(* Logix 5000 project; controller Heat_circuit_control Emulate 5570 rev 30.12; software revision 30.01 *)

TASK MainTask (continuous, watchdog 500 ms) : MainProgram

MODULES
   Local : Emulate 5570 (ICP 3, rev 30.12)
      HOA_Digital_module : 1756-IB16 (ICP 2, rev 3.1, Input RPI 20 ms)
      Alarm_digital_output : vendor 1 type 7 code 18 (ICP 4, rev 3.1, Output RPI 20 ms)
      Analog_Valve_control : vendor 1 type 10 code 114 (ICP 0, rev 2.1, Input RPI 100 ms)
      Analog_Temperature_Output : vendor 1 type 10 code 115 (ICP 1, rev 2.1, Output RPI 25 ms)
END_MODULES

VAR_GLOBAL   (* controller tags *)
   Auto_control : ALIAS FOR Local:2:I.Data.2;
   Hand_control : ALIAS FOR Local:2:I.Data.0;
   Off_control : ALIAS FOR Local:2:I.Data.1;
   Solenoid_Valve : ALIAS FOR Local:0:I.Ch1Data;
   Temperature_level : ALIAS FOR Local:1:O.Ch1Data;
END_VAR

PROGRAM MainProgram   (* main routine MainRoutine *)
VAR
   Alarm : ALIAS FOR Local:4:O.Data.1;
   alarm_on : BOOL;
   Alarm_reset : ALIAS FOR Local:4:O.Data.0;
   alarm_timer : TIMER := (PRE := 5000);
   auto : BOOL;
   auto_mode : BOOL;
   check_timer : TIMER := (PRE := 5000);
   checking_light : BOOL;
   close_bit : BOOL;
   count : COUNTER;
   danger_bit : BOOL;
   high_limit : REAL;
   HOA : DINT;
   low_point : REAL;
   Manual : BOOL;
   Notification : ALIAS FOR Local:4:O.Data.2;
   OFF : BOOL;
   ons : BOOL;
   ons_10 : BOOL;
   ons_2 : BOOL;
   ons_3 : BOOL;
   ons_9 : BOOL;
   open_bit : BOOL;
   Openning : REAL;
   Set_Point : REAL;
   Solenoid_Valve_1 : REAL;
   Sub_light : BOOL;
   Timer_wait : TIMER := (PRE := 5000);
   Timer_wait_2 : TIMER := (PRE := 5000);
   Total : REAL;
   transfer : REAL;
   TT : BOOL;
   TT_2 : BOOL;
   TT_3 : BOOL;
   TT_4 : BOOL;
   user_input : REAL;
   user_val : REAL;
   value : REAL;
   wait_timer : TIMER := (PRE := 5000);
   wait_timer_2 : TIMER := (PRE := 5000);
END_VAR

ROUTINE Alarm   (* ladder *)
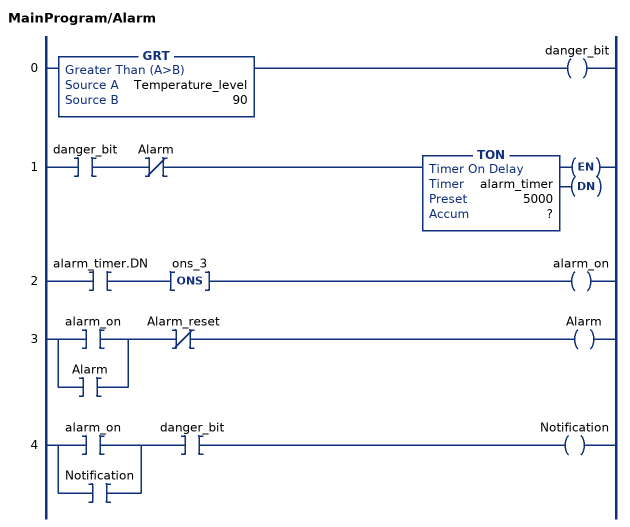
   0: GRT(Temperature_level,90)OTE(danger_bit);
   1: XIC(danger_bit)XIO(Alarm)TON(alarm_timer,?,?);
   2: XIC(alarm_timer.DN)ONS(ons_3)OTE(alarm_on);
   3: [XIC(alarm_on) ,XIC(Alarm) ]XIO(Alarm_reset)OTE(Alarm);
   4: [XIC(alarm_on) ,XIC(Notification) ]XIC(danger_bit)OTE(Notification);
END_ROUTINE

ROUTINE CONTROL   (* ladder *)
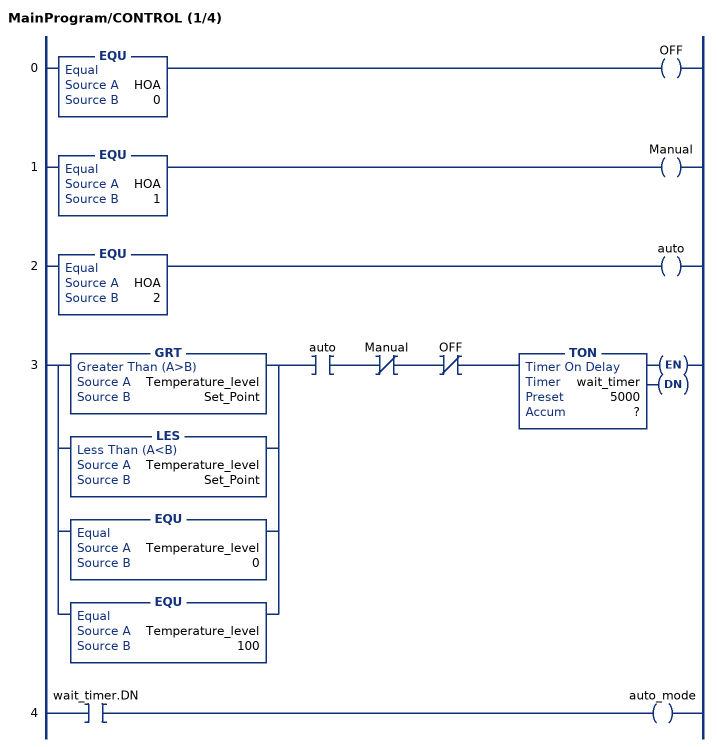
   0: EQU(HOA,0)OTE(OFF);
   1: EQU(HOA,1)OTE(Manual);
   2: EQU(HOA,2)OTE(auto);
   3: [GRT(Temperature_level,Set_Point) ,LES(Temperature_level,Set_Point) ,EQU(Temperature_level,0) ,EQU(Temperature_level,100) ]XIC(auto)XIO(Manual)XIO(OFF)TON(wait_timer,?,?);
   4: XIC(wait_timer.DN)OTE(auto_mode);
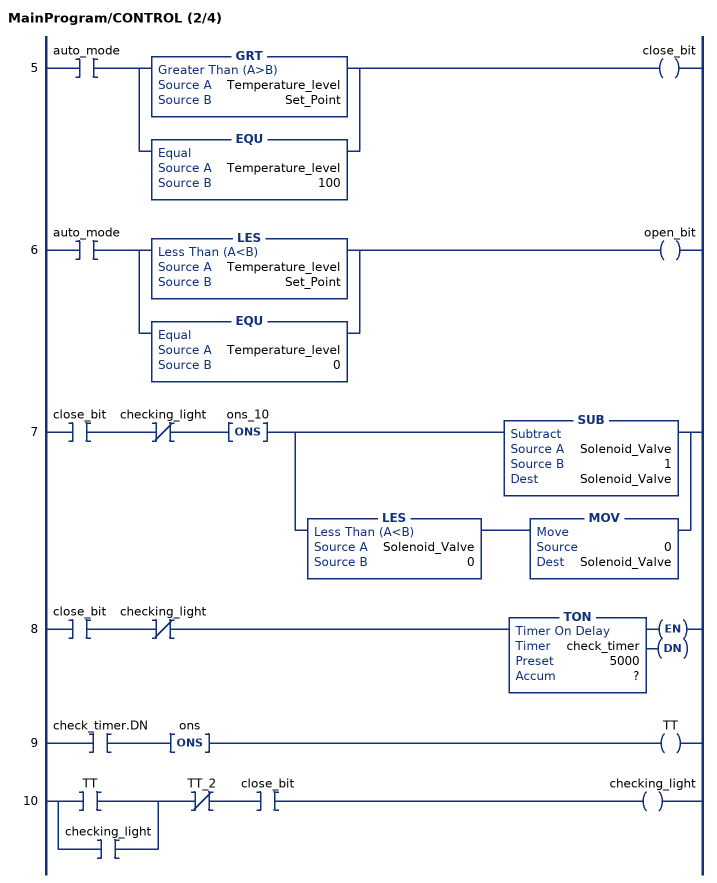
   5: XIC(auto_mode)[GRT(Temperature_level,Set_Point) ,EQU(Temperature_level,100) ]OTE(close_bit);
   6: XIC(auto_mode)[LES(Temperature_level,Set_Point) ,EQU(Temperature_level,0) ]OTE(open_bit);
   7: XIC(close_bit)XIO(checking_light)ONS(ons_10)[SUB(Solenoid_Valve,1,Solenoid_Valve) ,LES(Solenoid_Valve,0) MOV(0,Solenoid_Valve) ];
   8: XIC(close_bit)XIO(checking_light)TON(check_timer,?,?);
   9: XIC(check_timer.DN)ONS(ons)OTE(TT);
   10: [XIC(TT) ,XIC(checking_light) ]XIO(TT_2)XIC(close_bit)OTE(checking_light);
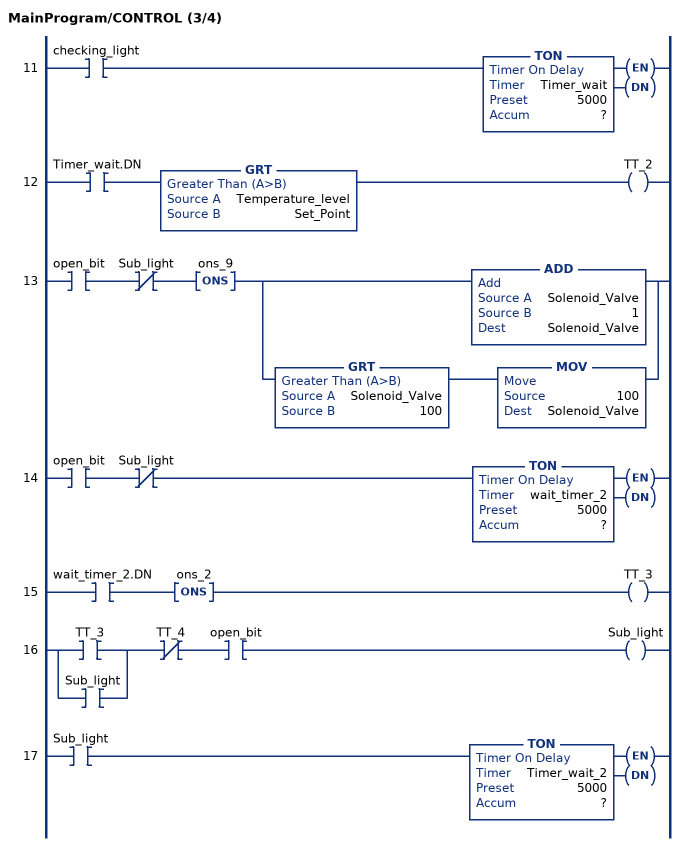
   11: XIC(checking_light)TON(Timer_wait,?,?);
   12: XIC(Timer_wait.DN)GRT(Temperature_level,Set_Point)OTE(TT_2);
   13: XIC(open_bit)XIO(Sub_light)ONS(ons_9)[ADD(Solenoid_Valve,1,Solenoid_Valve) ,GRT(Solenoid_Valve,100) MOV(100,Solenoid_Valve) ];
   14: XIC(open_bit)XIO(Sub_light)TON(wait_timer_2,?,?);
   15: XIC(wait_timer_2.DN)ONS(ons_2)OTE(TT_3);
   16: [XIC(TT_3) ,XIC(Sub_light) ]XIO(TT_4)XIC(open_bit)OTE(Sub_light);
   17: XIC(Sub_light)TON(Timer_wait_2,?,?);
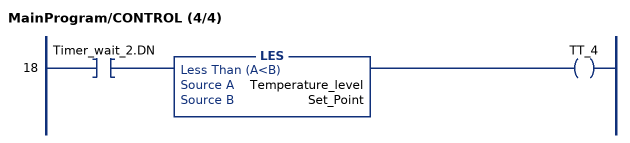
   18: XIC(Timer_wait_2.DN)LES(Temperature_level,Set_Point)OTE(TT_4);
END_ROUTINE

ROUTINE MainRoutine   (* ladder *)
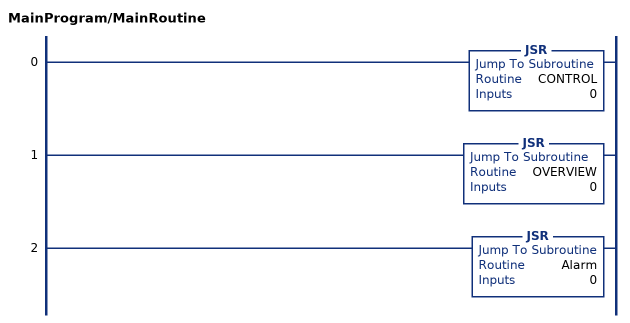
   0: JSR(CONTROL,0);
   1: JSR(OVERVIEW,0);
   2: JSR(Alarm,0);
END_ROUTINE

ROUTINE OVERVIEW   (* ladder *)
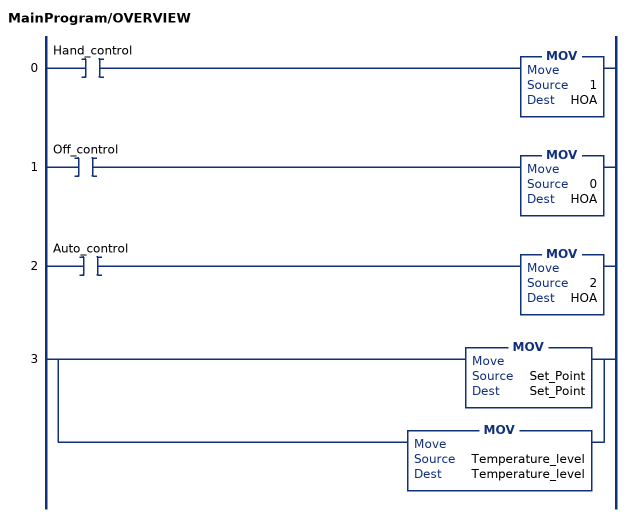
   0: XIC(Hand_control)MOV(1,HOA);
   1: XIC(Off_control)MOV(0,HOA);
   2: XIC(Auto_control)MOV(2,HOA);
   3: [MOV(Set_Point,Set_Point) ,MOV(Temperature_level,Temperature_level) ];
END_ROUTINE
END_PROGRAM
